// TIA Portal V16 export
// export: Created 2022-11-17T15:49:46.2611206Z, ExportSetting WithDefaults, DisplayName Totally Integrated Automation Portal, DisplayVersion V16 Update 6, DisplayName TIA Portal Version Control Interface, DisplayVersion V16 Update 2, DisplayName TIA Portal Openness, DisplayVersion V16 Update 6, DisplayName SINAMICS Startdrive Advanced, DisplayVersion V16 Update 5, DisplayName SINAMICS Startdrive G130, G150, S120, S150, SINAMICS MV, S210, DisplayVersion V16 Update 5, DisplayName SINAMICS Startdrive G110M, G120, G120C, G120D, G120P, G115D, DisplayVersion V16 Update 5, DisplayName STEP 7 Professional, DisplayVersion V16 Update 6, DisplayName STEP 7 Safety, DisplayVersion V16, DisplayName WinCC Advanced, DisplayVersion V16 Update 6
DATA_BLOCK "DB248_Program2"   // DB248
{ S7_Optimized_Access := 'FALSE' }
AUTHOR : Robopac
VERSION : 0.0
// stored: AutoNumber false, IsOnlyStoredInLoadMemory false, IsWriteProtectedInAS false
   VAR RETAIN
      Program2 { S7_SetPoint := 'True'} : "DatiProgramma";
   END_VAR
BEGIN
   Program2.Wrapping := TRUE;
   Program2.TopLenght := 500;
   Program2.TopRelease := 0;
   Program2.TopDown := 0;
   Program2.Top := 4;
   Program2.PressurePTime := 0;
   Program2.LifterTime := 0;
   Program2.RevOverContrast := 1;
   Program2.RopeEndCycle := 16#01;
   Program2.Spare4 := 16#01;
   Program2.RopeTime := 1500;
   Program2.RevOverClamp := 1;
   Program2.FilmForceFinalRev := 35;
   Program2.FilmPrestretchFinalRev := 100;
   Program2.ArmSpeed := 85;
   Program2.CarriageDown4Top := 500;
   Program2.TopDownTime := 1500;
   Program2.LapsUnderTop := 0;
   Program2.Spare6 := 0;
   Program2.Spare7 := 0;
   Program2.Spare8 := 0;
   Program2.Spare9 := 0;
   Program2.Spare10 := 0;
   Program2.Spare11 := 0;
   Program2.Spare12 := 0;
   Program2.Overlap0_1 := 0;
   Program2.Height1 := 180;
   Program2.Landmark1 := FALSE;
   Program2.Lifter1 := FALSE;
   Program2.SpareBit1H1 := FALSE;
   Program2.Airblower1 := TRUE;
   Program2.NextStep1 := TRUE;
   Program2.PressureP1 := TRUE;
   Program2.SpareByte2H1 := 16#00;
   Program2.Revolution1 := 1;
   Program2.RopeUnit1_1 := 16#01;
   Program2.RopeUnit1_2 := 16#01;
   Program2.FilmForce1 := 5;
   Program2.FilmPrestretch1 := 200;
   Program2.Spare3H1 := 0;
   Program2.Spare49 := 0;
   Program2.Spare50 := 0;
   Program2.Spare51 := 0;
   Program2.Spare52 := 0;
   Program2.Spare53 := 0;
   Program2.Overlap1_2 := 200;
   Program2.Height2 := -100;
   Program2.Landmark2 := TRUE;
   Program2.Lifter2 := FALSE;
   Program2.SpareBit1H2 := FALSE;
   Program2.Airblower2 := TRUE;
   Program2.NextStep2 := TRUE;
   Program2.PressureP2 := TRUE;
   Program2.SpareByte2H2 := 16#00;
   Program2.Revolution2 := 2;
   Program2.RopeUnit2_1 := 16#01;
   Program2.RopeUnit2_2 := 16#01;
   Program2.FilmForce2 := 20;
   Program2.FilmPrestretch2 := 200;
   Program2.Spare3H2 := 0;
   Program2.Spare54 := 0;
   Program2.Spare55 := 0;
   Program2.Spare56 := 0;
   Program2.Spare57 := 0;
   Program2.Spare58 := 0;
   Program2.Overlap2_3 := 200;
   Program2.Height3 := 80;
   Program2.Landmark3 := FALSE;
   Program2.Lifter3 := FALSE;
   Program2.SpareBit1H3 := FALSE;
   Program2.Airblower3 := TRUE;
   Program2.NextStep3 := TRUE;
   Program2.PressureP3 := TRUE;
   Program2.SpareByte2H3 := 16#00;
   Program2.Revolution3 := 2;
   Program2.RopeUnit3_1 := 16#01;
   Program2.RopeUnit3_2 := 16#01;
   Program2.FilmForce3 := 10;
   Program2.FilmPrestretch3 := 200;
   Program2.Spare3H3 := 0;
   Program2.Spare59 := 0;
   Program2.Spare60 := 0;
   Program2.Spare61 := 380;
   Program2.Spare62 := 2800;
   Program2.Spare63 := 0;
   Program2.Overlap3_4 := 200;
   Program2.Height4 := 120;
   Program2.Landmark4 := FALSE;
   Program2.Lifter4 := FALSE;
   Program2.SpareBit1H4 := FALSE;
   Program2.Airblower4 := TRUE;
   Program2.NextStep4 := TRUE;
   Program2.PressureP4 := TRUE;
   Program2.SpareByte2H4 := 16#00;
   Program2.Revolution4 := 2;
   Program2.RopeUnit4_1 := 16#02;
   Program2.RopeUnit4_2 := 16#02;
   Program2.FilmForce4 := 20;
   Program2.FilmPrestretch4 := 200;
   Program2.Spare3H4 := 0;
   Program2.Spare64 := 0;
   Program2.Spare65 := 0;
   Program2.Spare66 := 0;
   Program2.Spare67 := 0;
   Program2.Spare68 := 0;
   Program2.Overlap4_5 := 200;
   Program2.Height5 := 90;
   Program2.Landmark5 := FALSE;
   Program2.Lifter5 := FALSE;
   Program2.SpareBit1H5 := FALSE;
   Program2.Airblower5 := TRUE;
   Program2.NextStep5 := FALSE;
   Program2.PressureP5 := FALSE;
   Program2.SpareByte2H5 := 16#00;
   Program2.Revolution5 := 1;
   Program2.RopeUnit5_1 := 16#01;
   Program2.RopeUnit5_2 := 16#01;
   Program2.FilmForce5 := 20;
   Program2.FilmPrestretch5 := 200;
   Program2.Spare3H5 := 0;
   Program2.Spare69 := 0;
   Program2.Spare70 := 0;
   Program2.Spare71 := 0;
   Program2.Spare72 := 0;
   Program2.Spare73 := 0;
   Program2.Overlap5_6 := 300;
   Program2.Height6 := 120;
   Program2.Landmark6 := FALSE;
   Program2.Lifter6 := FALSE;
   Program2.SpareBit1H6 := FALSE;
   Program2.Airblower6 := TRUE;
   Program2.NextStep6 := FALSE;
   Program2.PressureP6 := FALSE;
   Program2.SpareByte2H6 := 16#00;
   Program2.Revolution6 := 1;
   Program2.RopeUnit6_1 := 16#01;
   Program2.RopeUnit6_2 := 16#01;
   Program2.FilmForce6 := 20;
   Program2.FilmPrestretch6 := 200;
   Program2.Spare3H6 := 0;
   Program2.Spare74 := 0;
   Program2.Spare75 := 0;
   Program2.Spare76 := 0;
   Program2.Spare77 := 0;
   Program2.Spare78 := 0;
   Program2.Overlap6_7 := 0;
   Program2.Height7 := 0;
   Program2.Landmark7 := FALSE;
   Program2.Lifter7 := FALSE;
   Program2.SpareBit1H7 := FALSE;
   Program2.Airblower7 := FALSE;
   Program2.NextStep7 := TRUE;
   Program2.PressureP7 := FALSE;
   Program2.SpareByte2H7 := 16#00;
   Program2.Revolution7 := 1;
   Program2.RopeUnit7_1 := 16#01;
   Program2.RopeUnit7_2 := 16#01;
   Program2.FilmForce7 := 0;
   Program2.FilmPrestretch7 := 100;
   Program2.Spare3H7 := 0;
   Program2.Spare79 := 0;
   Program2.Spare80 := 0;
   Program2.Spare81 := 0;
   Program2.Spare82 := 0;
   Program2.Spare83 := 0;
   Program2.Overlap7_8 := 0;
   Program2.Height8 := 0;
   Program2.Landmark8 := FALSE;
   Program2.Lifter8 := FALSE;
   Program2.SpareBit1H8 := FALSE;
   Program2.Airblower8 := FALSE;
   Program2.NextStep8 := TRUE;
   Program2.PressureP8 := FALSE;
   Program2.SpareByte2H8 := 16#00;
   Program2.Revolution8 := 1;
   Program2.RopeUnit8_1 := 16#01;
   Program2.RopeUnit8_2 := 16#01;
   Program2.FilmForce8 := 0;
   Program2.FilmPrestretch8 := 100;
   Program2.Spare3H8 := 0;
   Program2.Spare84 := 0;
   Program2.Spare85 := 0;
   Program2.Spare86 := 0;
   Program2.Spare87 := 0;
   Program2.Spare88 := 0;
   Program2.Overlap8_9 := 0;
   Program2.Height9 := 0;
   Program2.Landmark9 := FALSE;
   Program2.Lifter9 := FALSE;
   Program2.SpareBit1H9 := FALSE;
   Program2.Airblower9 := FALSE;
   Program2.NextStep9 := TRUE;
   Program2.PressureP9 := FALSE;
   Program2.SpareByte2H9 := 16#00;
   Program2.Revolution9 := 1;
   Program2.RopeUnit9_1 := 16#01;
   Program2.RopeUnit9_2 := 16#01;
   Program2.FilmForce9 := 0;
   Program2.FilmPrestretch9 := 100;
   Program2.Spare3H9 := 0;
   Program2.Spare89 := 0;
   Program2.Spare90 := 0;
   Program2.Spare91 := 0;
   Program2.Spare92 := 0;
   Program2.Spare93 := 0;
   Program2.Overlap9_10 := 0;
   Program2.Height10 := 0;
   Program2.Landmark10 := FALSE;
   Program2.Lifter10 := FALSE;
   Program2.SpareBit1H10 := FALSE;
   Program2.Airblower10 := FALSE;
   Program2.NextStep10 := FALSE;
   Program2.PressureP10 := FALSE;
   Program2.SpareByte2H10 := 16#00;
   Program2.Revolution10 := 1;
   Program2.RopeUnit10_1 := 16#01;
   Program2.RopeUnit10_2 := 16#01;
   Program2.FilmForce10 := 0;
   Program2.FilmPrestretch10 := 100;
   Program2.Spare3H10 := 0;
   Program2.Spare94 := 0;
   Program2.Spare95 := 0;
   Program2.Spare96 := 0;
   Program2.Spare97 := 0;
   Program2.Spare98 := 0;
   Program2.Overlap10_11 := 0;
   Program2.Height11 := 0;
   Program2.Landmark11 := FALSE;
   Program2.Lifter11 := FALSE;
   Program2.SpareBit1H11 := FALSE;
   Program2.Airblower11 := FALSE;
   Program2.NextStep11 := TRUE;
   Program2.PressureP11 := FALSE;
   Program2.SpareByte2H11 := 16#00;
   Program2.Revolution11 := 1;
   Program2.RopeUnit11_1 := 16#01;
   Program2.RopeUnit11_2 := 16#01;
   Program2.FilmForce11 := 0;
   Program2.FilmPrestretch11 := 100;
   Program2.Spare3H11 := 0;
   Program2.Spare99 := 0;
   Program2.Spare100 := 0;
   Program2.Spare101 := 0;
   Program2.Spare102 := 0;
   Program2.Spare103 := 0;
   Program2.Overlap11_12 := 0;
   Program2.Height12 := 0;
   Program2.Landmark12 := FALSE;
   Program2.Lifter12 := FALSE;
   Program2.SpareBit1H12 := FALSE;
   Program2.Airblower12 := FALSE;
   Program2.NextStep12 := FALSE;
   Program2.PressureP12 := FALSE;
   Program2.SpareByte2H12 := 16#00;
   Program2.Revolution12 := 1;
   Program2.RopeUnit12_1 := 16#01;
   Program2.RopeUnit12_2 := 16#01;
   Program2.FilmForce12 := 0;
   Program2.FilmPrestretch12 := 100;
   Program2.Spare3H12 := 0;
   Program2.Spare104 := 0;
   Program2.Spare105 := 0;
   Program2.Spare106 := 0;
   Program2.Spare107 := 0;
   Program2.Spare108 := 0;
END_DATA_BLOCK
